TYPE st_Wifi :
STRUCT
	WifiClienModeStatus		:	eWifiStatus;
	WifiAPModeStatus		:	eWifiStatus;
	WifiApNumberOfClients	:	Uint;
END_STRUCT
END_TYPE

(* stored: Version 1.1.0.1, ProductVersion 3.1.4026.18
   DUT st_Wifi: Id {42e7f11a-6ea3-45da-9890-c7ad4bd5f487} *)
